Universal Robots PolyScope program: prueba.urp

Program drill291217_1952 (createdIn=3.4.5.437 lastSavedIn=3.4.5.437 directory=/programs/usbdisk installation=default robotSerialNumber=2017307081)
Calibrated DH parameters: a=[0.000065, -0.609605, -0.569684, 0.000059, 0.000099, 0]; d=[0.128194, 4.336054, 1.236291, -5.409118, 0.11576, 0.092314]; alpha=[1.570898, -0.013944, -0.007792, 1.5711, -1.5712, 0]; deltaTheta=[0.006367, -0.089589, 0.029531, 0.074964, 0.034815, -0.025455]
BeforeStart
  MoveJ speed 60 deg/s, acceleration 80 deg/s^2 (useActiveTCP=false) tcp=TCP_2
    Waypoint Waypoint_1: TCP in base x=21.821 y=242.698 z=804.588 mm, rx=-2.915 ry=1.1275 rz=0.0621 rad; joints [180, -46.802, -93.569, -128.691, 86.442, 135] deg; flange x=-132.819 y=156.008 z=854.047 mm, rx=-2.915 ry=1.1274 rz=0.0621 rad
  conn := False
  contador := 1
  origen := get_actual_tcp_pose()
Robot Program (runOnlyOnce=false motionType=MoveJ speed=1.047198 acceleration=1.396263 useActiveTCP=false)
  Loop While (checkContinuously=false) expression=conn≟ False
    conn := socket_open("192.168.10.20",3000)
  Pallet pattern(dimensionality=Square firstAxisCount=2 secondAxisCount=3 thirdAxisCount=5 motionType=MoveL speed=0.25 acceleration=1.2 useActiveTCP=false, counterVariable(name=cnt_1, initializeExpression=0), patternPoseVariable(name=pose_1), feature=Base, children(Waypoint(type=Fixed name=a1st_Corner_1, position(joints=4.118790680570999, -1.1650667232594119, -1.5046604681423776, -2.064424738363112, 1.4910444549653672, 3.3347764297117344 pose=-0.18506112197563362, -0.13831893089874014, 0.8136686768505219, -2.9149189170158607, 1.1274601196302712, 0.0621328068109231), poseInFeatureCoordinates=[-0.185061, -0.138319, 0.813669, -2.914919, 1.12746, 0.062133], outputFlangePose=[-0.339657, -0.225015, 0.863153, -2.91498, 1.127475, 0.06208]), Waypoint(type=Fixed name=a2nd_Corner_1, position(joints=3.0173065554847764, -1.1287651824094276, -1.5467624160193143, -2.0171261926526647, 1.5080532911858793, 2.2323976591195267 pose=-0.18502672006388193, 0.2845138717082553, 0.80632867827917, -2.9150027221100197, 1.1272927335330698, 0.062097882733016654), poseInFeatureCoordinates=[-0.185027, 0.284514, 0.806329, -2.915003, 1.127293, 0.062098], outputFlangePose=[-0.339657, 0.197816, 0.855762, -2.91498, 1.127475, 0.06208]), Waypoint(type=Fixed name=a3rd_Corner_1, position(joints=3.0173158268909543, -1.1015408347234459, -1.6340938501223166, -1.9570027076395515, 1.5082549266276795, 2.231841892250847 pose=-0.1850423120051651, 0.28451222142269467, 0.7679767683501497, -2.9150933640644485, 1.1273494152376073, 0.06213147539161546), poseInFeatureCoordinates=[-0.185042, 0.284512, 0.767977, -2.915093, 1.127349, 0.062131], outputFlangePose=[-0.339657, 0.197816, 0.817427, -2.91498, 1.127475, 0.06208]), Waypoint(type=Fixed name=a4th_Corner_1, position(joints=4.124959130921647, -1.1365499826462298, -1.6079587282217265, -1.9898716825047673, 1.4912480962655819, 3.3402778846434416 pose=-0.18505481868755233, -0.14260773960947615, 0.7679522114623871, -2.9149255897909176, 1.1274867033547258, 0.06198546347264506), poseInFeatureCoordinates=[-0.185055, -0.142608, 0.767952, -2.914926, 1.127487, 0.061985], outputFlangePose=[-0.339657, -0.229279, 0.817427, -2.91498, 1.127475, 0.06208]))); actionSequence(name=PalletSequence motionType=MoveL speed=0.25 acceleration=1.2 useActiveTCP=false, anchorWaypoint(type=Fixed name=PatternPoint_1, position(joints=4.16423677147252, -1.081988811079853, -1.5196656321692084, -2.083411083527203, 1.5426363635044549, 1.8131091385151614 pose=-0.17500620268307482, -0.029864776507154883, 0.8018281004608351, 2.846518819290686, 1.252680709352249, -0.04482889806087609), poseInFeatureCoordinates=[-0.175006, -0.029865, 0.801828, 2.846519, 1.252681, -0.044829], outputFlangePose=[-0.293735, -0.19065, 0.880317, 2.846595, 1.252497, -0.044902]), feature=Base, children(Waypoint(type=Fixed name=Approach_1, position(joints=4.16423677147252, -1.081988811079853, -1.5196656321692084, -2.083411083527203, 1.5426363635044549, 1.8131091385151614 pose=-0.17501592179798203, -0.029886752142520286, 0.8018303729568981, 2.8465872998729034, 1.2527285167879534, -0.04480737981762656), poseInFeatureCoordinates=[-0.175016, -0.029887, 0.80183, 2.846587, 1.252729, -0.044807], outputFlangePose=[-0.293735, -0.19065, 0.880317, 2.846595, 1.252497, -0.044902]), Waypoint=PatternPoint_1, Set(type=NoAction), Wait(type=Sleep, waitTime=3), CallSubProgram(subprogram(name=Trigger keepSynchronizedWithDisk=false trackProgramExecution=false, children(Script(type=Line, expression=socket_send_string("trigger_on")), Script(type=Line, expression=socket_send_byte(0)), Wait(type=Sleep, waitTime=0.5), Script(type=Line, expression=socket_send_string("trigger_off")), Script(type=Line, expression=socket_send_byte(0)), Wait(type=Sleep, waitTime=0.5), Assignment(valueSource=Expression, variable(name=Data), expression=socket_read_ascii_float(9))))), Assignment(valueSource=Expression, variable(name=cantidad), expression=Data[1]), If(type=If checkContinuously=false, expression=cantidad≠0, children(Loop(type=While checkContinuously=false, expression=contador≤cantidad, children(Assignment(valueSource=Expression, variable(name=Xfoto), expression=-Data[2*contador]), Assignment(valueSource=Expression, variable(name=Yfoto), expression=-Data[(2*contador+1)]), Assignment(valueSource=Expression, variable(name=pCamara), expression=get_actual_tcp_pose()), Set(type=NoAction, tcp=TCP_1), Assignment(valueSource=Expression, variable(name=pTaladro), expression=get_actual_tcp_pose()), Assignment(valueSource=Expression, variable(name=var_1), expression=pose_trans(pCamara,pTaladro)), Move(motionType=MoveJ speed=1.047198 acceleration=1.396263 useActiveTCP=false, tcp=TCP_1, children(Waypoint(type=Variable name=Waypoint, variable=var_1))), SuppressedNode(suppressedNode(valueSource=Expression, variable(name=delta), expression=pose_sub(pCamara,pTaladro))), SuppressedNode(suppressedNode(valueSource=Expression, variable(name=offset), expression=pose_add(pTaladro,delta))), SuppressedNode(suppressedNode(valueSource=Expression, variable(name=punto), expression=p[0,Xfoto,Yfoto,0,0,0])), SuppressedNode(suppressedNode(motionType=MoveL speed=0.25 acceleration=1.2 useActiveTCP=true, feature=Base, children(Waypoint(type=Variable name=Waypoint, variable=pCamara)))), SuppressedNode(suppressedNode(type=Sleep, waitTime=1)), SuppressedNode(suppressedNode(valueSource=Expression, variable(name=deltaoff), expression=pose_sub(offset,punto))), SuppressedNode(suppressedNode(motionType=MoveJ speed=1.047198 acceleration=1.396263 useActiveTCP=true, children(Waypoint(type=Variable name=Waypoint, variable=deltaoff), Wait(type=Sleep, waitTime=30)))), Assignment(valueSource=Expression, variable=contador, expression=contador+1))))), Set(type=NoAction, tcp=TCP_2), Waypoint(type=Fixed name=Exit_1, position(joints=4.16423677147252, -1.081988811079853, -1.5196656321692084, -2.083411083527203, 1.5426363635044549, 1.8131091385151614 pose=-0.1750297120850819, -0.02989601432756092, 0.8018258722096436, 2.8465869064362987, 1.2527086328217287, -0.04479713692533929), poseInFeatureCoordinates=[-0.17503, -0.029896, 0.801826, 2.846587, 1.252709, -0.044797], outputFlangePose=[-0.293735, -0.19065, 0.880317, 2.846595, 1.252497, -0.044902])))
    Pattern -> pattern
    AnchoredSequence -> PalletSequence
SubProgram -> Trigger
